# EPICS substitutions: iocs/ni9144-3modules/ni3modApp/Db/ni9234.substitutions
file MASTER.template
{
{DEVICE="RJQ35657-ECAT-01", PORT="MASTER0", SCAN="I/O Intr"}
}
file NI944.template
{
{DEVICE="RJQ35657-ECAT-02", PORT="NI0", SCAN=".1 second"}
}
file gadc.template
{
pattern {DEVICE, PORT, SCAN, SAMPLES, CHANNEL}
{RJQ35657-ECAT-02, NI0, ".1 second", 1000000, 1}
}
